Staubli VAL3: motionControl.pgx

public program motionControl()
  local MotionBuffer l_mTrajPt
  local bool l_bFlag
  local MotionBuffer l_motion
  local num l_nTime
  local bool l_bStopAndClean
begin
  nMoveId = -1

  while (true)
    // check connection status, and whether to stop motion
    if (nDataIn == 1 and nDataOut == 1 and bStopNow == false)

      nMotionProgress = getMoveId()

      // process trajectory point from trajectory buffer
      if (libTrajPtBuffer:nElems > 4)
        call libTrajPtBuffer:pop(l_mTrajPt, l_bFlag)
        if (l_bFlag)
          nPtsPopped = nPtsPopped + 1
          call libMoveBuffer:push(l_mTrajPt, l_bFlag)
          if (l_bFlag == false)
            //nMovePts = nMovePts + 1
          endIf
        endIf
      endIf

      // process motion command from move buffer
      // move buffer should have elements previously interpolated
      // to ensure they are 4 ms apart
      if (libMoveBuffer:nElems > 6)
        call libMoveBuffer:pop(l_motion, l_bFlag)
        if (l_bFlag)
          nMovePts = nMovePts + 1
//          if ((nMotionProgress-nMoveId) > 0.0)
//            nMoveId = movej(l_motion.jJointRx, tTool, l_motion.mDesc)
//            waitEndMove()
//            nMotionProgress = getMoveId()
//            // if this is the last motion command, call waitEndMove()
//            // to ensure point is reached
//            if (l_motion.nSequence == -1)
//              waitEndMove()
//            endIf
//          endIf
        endIf
      endIf
    else
      // stop immediately -- resetMotion() also resets moveId
      resetMotion()
      // clear buffers
      call libTrajPtBuffer:clear()
      call libMoveBuffer:clear()
      bStopNow = false

      // debug
      nPtsPopped = 0
      nMovePts = 0
    endIf

    // sequence task
    delay(0)
  endWhile
end
